FUNCTION_BLOCK FB_StateOpened
VAR_IN_OUT
	stAxis  	: ARRAY [GVL.cXP .. GVL.cXM] OF ST_AxisGroup;	
	bTopEntry	: BOOL;
END_VAR
VAR
	//state-machine
	nCurrentState	: INT;
	nNextState		: INT;
	
END_VAR


IF bTopEntry = TRUE THEN
	bTopEntry := FALSE;
	nNextState := 1200;
END_IF	
nCurrentState := nNextState;

CASE nCurrentState OF
	1200:
		stAxis[GVL.cXP].bBrake := GVL.cBrakeOn;
		stAxis[GVL.cXP].bBrake := GVL.cBrakeOn;


END_CASE

END_FUNCTION_BLOCK

(* stored: Version 1.1.0.1, ProductVersion 3.1.4022.18
   POU FB_StateOpened: Id {596682f8-87ed-401d-9eb9-43883efdf49e}, SpecialFunc None *)
